TYPE ST_Error :
STRUCT
	Active : BOOL := FALSE;
	Label : STRING(Param_Error.LABEL_LEN);
	Message : STRING(Param_Error.MESSAGE_LEN);
	Priority : E_ErrorPriority := E_ErrorPriority.Diagnostic;
END_STRUCT
END_TYPE

(* stored: Version 1.1.0.1, ProductVersion 3.1.4024.12
   DUT ST_Error: Id {bb9261a5-54e4-4675-87c5-c8ae85697e7d} *)
